FUNCTION_BLOCK MyCalculatorClass
VAR
END_VAR

METHOD Divide : INT
VAR_INPUT
	x : INT;
	y : INT;
END_VAR
IF y <> 0 THEN
	Divide := x/y;
ELSE
	Divide := -1;
END_IF
END_METHOD

END_FUNCTION_BLOCK

(* stored: Version 1.1.0.1, ProductVersion 3.1.4024.13
   POU MyCalculatorClass: Id {e86cfbde-ef3c-4c6f-af9b-c9b3d4bba912}, SpecialFunc None
   Method Divide: Id {22f95054-f08a-40f5-9e5b-77f39478afb5} *)
